// TIA Portal V17 export
// export: Created 2025-04-22T12:08:40.6512098Z, ExportSetting WithDefaults, DisplayName Totally Integrated Automation Portal, DisplayVersion V17 Update 8, DisplayName TIA Portal Openness, DisplayVersion V17 Update 8, DisplayName TIA Portal Version Control Interface, DisplayVersion V17, DisplayName SINAMICS Startdrive Advanced, DisplayVersion V17 SP2, DisplayName SINAMICS Startdrive G110M, G120, G120C, G120D, G120P, G115D, DisplayVersion V17 SP2, DisplayName SINAMICS Startdrive G130, G150, S120, S150, SINAMICS MV, S210, DisplayVersion V17 SP2, DisplayName STEP 7 Professional, DisplayVersion V17 Update 8, DisplayName SINUMERIK ONE STEP 7 Toolbox, DisplayVersion V17 Update 12, DisplayName SINUMERIK 840D sl STEP 7 Toolbox, DisplayVersion V17 Update 12, DisplayName STEP 7 Safety, DisplayVersion V17 Update 6, DisplayName WinCC Advanced / Unified PC, DisplayVersion V17 Update 8
FUNCTION "FC1701_KELLER_ASPIRATION_CONTROL" : Void   // FC1701, LAD
{ S7_Optimized_Access := 'TRUE' }
VERSION : 0.1
// stored: AutoNumber false, IsIECCheckEnabled false, SetENOAutomatically false, UDAEnableTagReadback false
   VAR CONSTANT
      FC_NUMBER : DInt := 1701;
   END_VAR
BEGIN

REGION Network 1: <<<<<<<<<<<<<<<<<<<< ASPIRATION CONTROL >>>>>>>>>>>>>>>>>>>>
END_REGION

REGION Network 2: CALL FB1701 KELLER ASPIRATION CONTROL
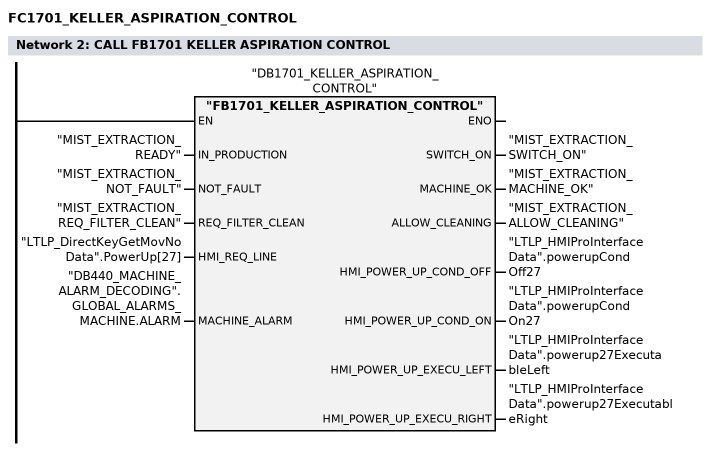
   RUNG wire#powerrail
      "DB1701_KELLER_ASPIRATION_CONTROL"(IN_PRODUCTION := "MIST_EXTRACTION_READY", NOT_FAULT := "MIST_EXTRACTION_NOT_FAULT", REQ_FILTER_CLEAN := "MIST_EXTRACTION_REQ_FILTER_CLEAN", HMI_REQ_LINE := "LTLP_DirectKeyGetMovNoData".PowerUp[27], MACHINE_ALARM := "DB440_MACHINE_ALARM_DECODING".GLOBAL_ALARMS_MACHINE.ALARM, SWITCH_ON => "MIST_EXTRACTION_SWITCH_ON", MACHINE_OK => "MIST_EXTRACTION_MACHINE_OK", ALLOW_CLEANING => "MIST_EXTRACTION_ALLOW_CLEANING", HMI_POWER_UP_COND_OFF => "LTLP_HMIProInterfaceData".powerupCondOff27, HMI_POWER_UP_COND_ON => "LTLP_HMIProInterfaceData".powerupCondOn27, HMI_POWER_UP_EXECU_LEFT => "LTLP_HMIProInterfaceData".powerup27ExecutableLeft, HMI_POWER_UP_EXECU_RIGHT => "LTLP_HMIProInterfaceData".powerup27ExecutableRight)
   END_RUNG
   // the same network as SCL:
   "DB1701_KELLER_ASPIRATION_CONTROL"(IN_PRODUCTION := "MIST_EXTRACTION_READY",   // "FB1701_KELLER_ASPIRATION_CONTROL"
                           NOT_FAULT := "MIST_EXTRACTION_NOT_FAULT",
                           REQ_FILTER_CLEAN := "MIST_EXTRACTION_REQ_FILTER_CLEAN",
                           HMI_REQ_LINE := "LTLP_DirectKeyGetMovNoData".PowerUp[27],
                           MACHINE_ALARM := "DB440_MACHINE_ALARM_DECODING".GLOBAL_ALARMS_MACHINE.ALARM,
                           SWITCH_ON => "MIST_EXTRACTION_SWITCH_ON",
                           MACHINE_OK => "MIST_EXTRACTION_MACHINE_OK",
                           ALLOW_CLEANING => "MIST_EXTRACTION_ALLOW_CLEANING",
                           HMI_POWER_UP_COND_OFF => "LTLP_HMIProInterfaceData".powerupCondOff27,
                           HMI_POWER_UP_COND_ON => "LTLP_HMIProInterfaceData".powerupCondOn27,
                           HMI_POWER_UP_EXECU_LEFT => "LTLP_HMIProInterfaceData".powerup27ExecutableLeft,
                           HMI_POWER_UP_EXECU_RIGHT => "LTLP_HMIProInterfaceData".powerup27ExecutableRight);
END_REGION
END_FUNCTION
